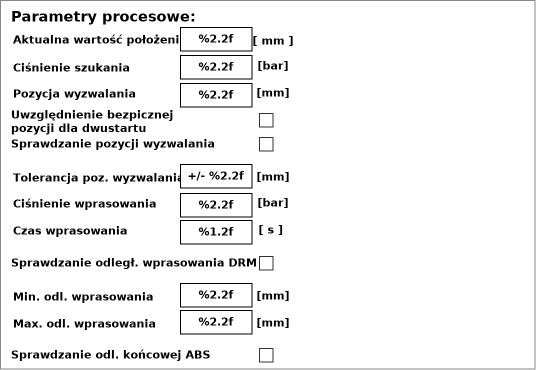
VISUALIZATION vSonicPress_SubSettings  // 536x370
VAR_IN_OUT
	fbMachine:fbSonicPress;
	stTestParams:stSonicPress_TestParams;
END_VAR
    Label (10,56 169x24), "Ciśnienie szukania"
    Rectangle (180,55 72x24), "%2.2f", text variable: stTestParams.rSearchPressure, input disabled if: NOT GVL.fbUserLogin.bPermissionGranted
        OnMouseClick: write the text variable via Default, min 0.2, max 3
    Label (252,54 42x24), "[bar]"
    Label (10,219 169x24), "Czas wprasowania"
    Rectangle (180,220 72x24), "%1.2f", text variable: stTestParams.rPressTime, input disabled if: NOT GVL.fbUserLogin.bPermissionGranted
        OnMouseClick: write the text variable via Default, min 0.2, max 9.9, title 'Press time'
    Label (252,218 42x24), "[ s ]"
    Label (10,28 169x24), "Aktualna wartość położenia"
    Rectangle (180,27 72x24), "%2.2f", text variable: fbMachine.fbPositionMeasure.rOutFiltered
    Label (252,29 42x24), "[ mm ]"
    Label (8,132 226x24), "Sprawdzanie pozycji wyzwalania"
    Checkbox (257,131 26x26), variable: stTestParams.bCheckTriggerPos, input disabled if: NOT GVL.fbUserLogin.bPermissionGranted
    Label (10,192 169x24), "Ciśnienie wprasowania"
    Rectangle (180,193 72x24), "%2.2f", text variable: stTestParams.rPressPressure, input disabled if: NOT GVL.fbUserLogin.bPermissionGranted
        OnMouseClick: write the text variable via Default, min 0.5, max 6, title 'Press pressure'
    Label (252,191 42x24), "[bar]"
    Label (252,81 42x24), "[mm]"
    Label (10,82 169x24), "Pozycja wyzwalania"
    Rectangle (180,83 72x24), "%2.2f", text variable: stTestParams.rTriggerPos, input disabled if: NOT GVL.fbUserLogin.bPermissionGranted
        OnMouseClick: write the text variable via Default, min 1, max 30, title 'Trigger position'
    Label (252,165 42x24), "[mm]"
    Label (10,166 169x24), "Tolerancja poz. wyzwalania"
    Rectangle (180,164 72x24), "+/- %2.2f", text variable: stTestParams.rTriggerPosMaxDeviation, input disabled if: NOT GVL.fbUserLogin.bPermissionGranted
        OnMouseClick: write the text variable via Default, min 0.01, max 10, title 'Trigger max deviation'
    Label (8,251 240x24), "Sprawdzanie odległ. wprasowania DRM"
    Checkbox (257,250 26x26), variable: stTestParams.bCheckPressLength, input disabled if: NOT GVL.fbUserLogin.bPermissionGranted
    Label (10,285 169x24), "Min. odl. wprasowania"
    Label (252,284 42x24), "[mm]"
    Rectangle (180,283 72x24), "%2.2f", text variable: stTestParams.rMinPressLength, input disabled if: NOT GVL.fbUserLogin.bPermissionGranted
        OnMouseClick: write the text variable via Default, min 0.01, max 30.0, title 'Min press length'
    Label (10,312 169x24), "Max. odl. wprasowania"
    Label (252,311 42x24), "[mm]"
    Rectangle (180,310 72x24), "%2.2f", text variable: stTestParams.rMaxPressLength, input disabled if: NOT GVL.fbUserLogin.bPermissionGranted
        OnMouseClick: write the text variable via Default, min 0.01, max 30, title 'Max press length'
    Label (8,343 226x24), "Sprawdzanie odl. końcowej ABS"
    Checkbox (257,342 26x26), variable: stTestParams.bCheckEndPos, input disabled if: NOT GVL.fbUserLogin.bPermissionGranted
    Label (8,0 271x33), "Parametry procesowe:"
    Checkbox (257,107 26x26), variable: stTestParams.bUseOnlyStartEndVerification, input disabled if: NOT GVL.fbUserLogin.bPermissionGranted
    Label (8,104 225x35), "Uwzględnienie bezpicznej pozycji dla dwustartu"
END_VISUALIZATION

(* stored: Version 1.1.0.1, ProductVersion 3.1.4024.13
   Visu vSonicPress_SubSettings: Id {24351efc-8e56-47e6-8588-411dd098ba71} *)
